TYPE ST_CNCG159VG :
STRUCT
	sTarget: STRING(95);
	dValue: DINT;
END_STRUCT
END_TYPE

(* stored: Version 1.1.0.1, ProductVersion 3.1.0.17
   DUT ST_CNCG159VG: Id {9934803f-8061-44a5-b78e-61898006163d} *)
